TYPE ST_AlarmHistory :
STRUCT
    sTime		: STRING(255);
	sType		: E_Alarms := E_Alarms.Vazio;
	sDate		: STRING(255);
	abType		: DINT;	
    nEventId  	: INT;
    sMessage  	: STRING(255) := '';
END_STRUCT
END_TYPE

(* stored: Version 1.1.0.1
   DUT ST_AlarmHistory: Id {8a14a77e-92d1-4f79-92bd-adbe73675153} *)
